// SIMATIC S7-200 SMART project (STEP 7-Micro/WIN SMART), CPU SR40

ORGANIZATION_BLOCK 主程序:OB1
TITLE=程序注释
BEGIN
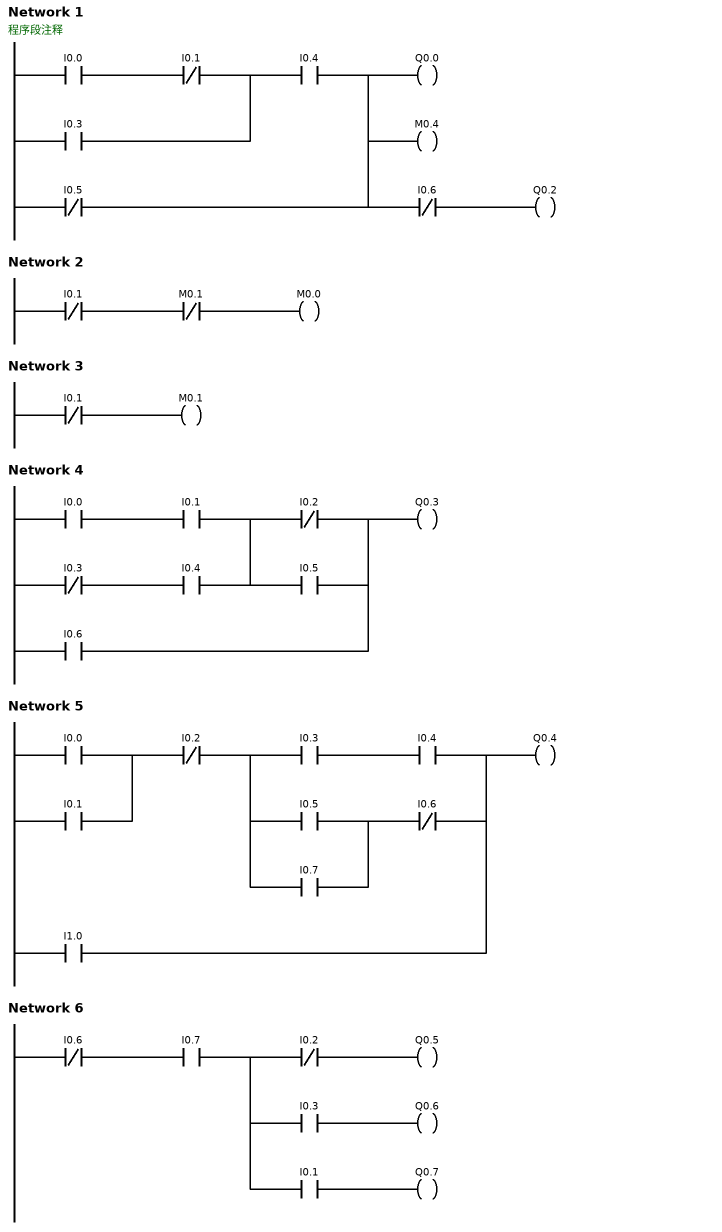
Network 1
// 程序段注释
LD     I0.0
AN     I0.1
O      I0.3
A      I0.4
ON     I0.5
=      Q0.0
=      M0.4
AN     I0.6
=      Q0.2
Network 2
LDN    I0.1
AN     M0.1
=      M0.0
Network 3
LDN    I0.1
=      M0.1
Network 4
LD     I0.0
A      I0.1
LDN    I0.3
A      I0.4
OLD
LDN    I0.2
O      I0.5
ALD
O      I0.6
=      Q0.3
Network 5
LD     I0.0
O      I0.1
AN     I0.2
LD     I0.3
A      I0.4
LD     I0.5
O      I0.7
AN     I0.6
OLD
ALD
O      I1.0
=      Q0.4
Network 6
LDN    I0.6
A      I0.7
LPS
AN     I0.2
=      Q0.5
LRD
A      I0.3
=      Q0.6
LPP
A      I0.1
=      Q0.7
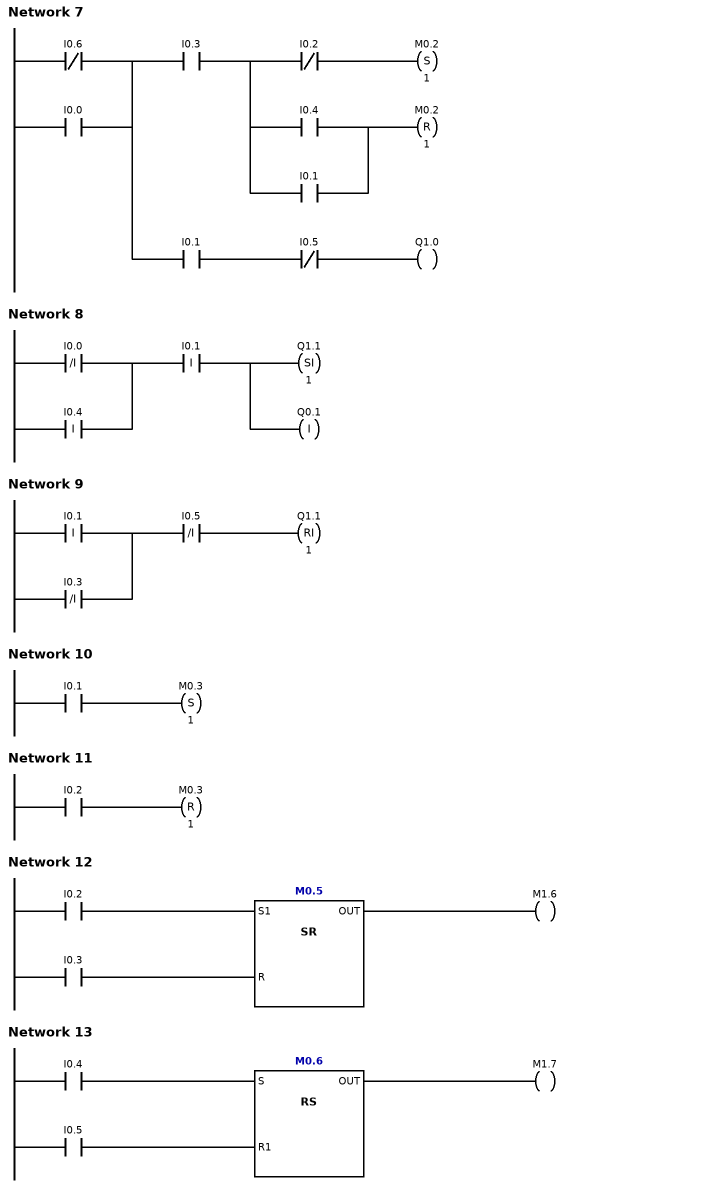
Network 7
LDN    I0.6
O      I0.0
LPS
A      I0.3
LPS
AN     I0.2
S      M0.2, 1
LPP
LD     I0.4
O      I0.1
ALD
R      M0.2, 1
LPP
A      I0.1
AN     I0.5
=      Q1.0
Network 8
LDNI   I0.0
OI     I0.4
AI     I0.1
SI     Q1.1, 1
=I     Q0.1
Network 9
LDI    I0.1
ONI    I0.3
ANI    I0.5
RI     Q1.1, 1
Network 10
LD     I0.1
S      M0.3, 1
Network 11
LD     I0.2
R      M0.3, 1
Network 12
LD     I0.2
LD     I0.3
NOT
A      M0.5
OLD
=      M0.5
=      M1.6
Network 13
LD     I0.4
LD     I0.5
NOT
LPS
A      M0.6
=      M0.6
LPP
ALD
O      M0.6
=      M0.6
=      M1.7
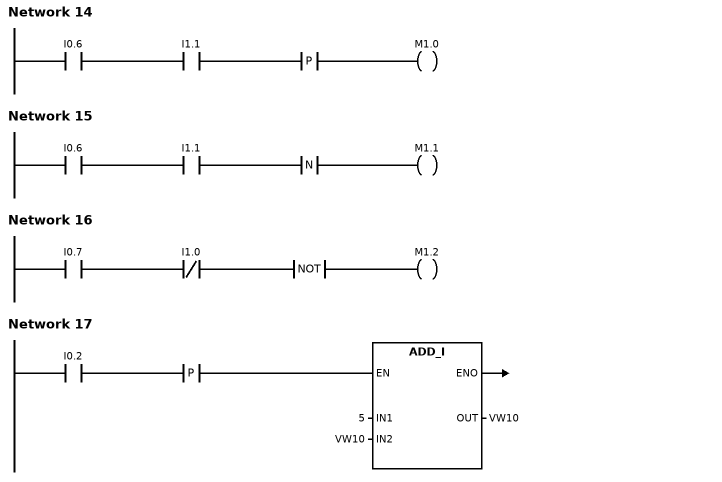
Network 14
LD     I0.6
A      I1.1
EU
=      M1.0
Network 15
LD     I0.6
A      I1.1
ED
=      M1.1
Network 16
LD     I0.7
AN     I1.0
NOT
=      M1.2
Network 17
LD     I0.2
EU
+I     5, VW10
END_ORGANIZATION_BLOCK
